// TIA Portal V17 export
// export: Created 2024-09-03T21:55:01.6127892Z, ExportSetting WithDefaults, DisplayName Totally Integrated Automation Portal, DisplayVersion V17 Update 7, DisplayName TIA Portal Openness, DisplayVersion V17 Update 7, DisplayName TIA Portal Version Control Interface, DisplayVersion V17, DisplayName SINAMICS Startdrive Advanced, DisplayVersion V17 SP2, DisplayName SINAMICS Startdrive G110M, G120, G120C, G120D, G120P, G115D, DisplayVersion V17 SP2, DisplayName SINAMICS Startdrive G130, G150, S120, S150, SINAMICS MV, S210, DisplayVersion V17 SP2, DisplayName STEP 7 Professional, DisplayVersion V17 Update 7, DisplayName STEP 7 Safety, DisplayVersion V17 Update 6, DisplayName WinCC Advanced / Unified PC, DisplayVersion V17 Update 7
DATA_BLOCK "IJC_DB"   // DB800
VERSION : 0.1
// stored: AutoNumber false, DBAccessibleFromOPCUA true, DBAccessibleFromWebserver true, InstanceOfName FB_IJC, InstanceOfType FB
"FB_IJC"
   // VAR
   //    MSG { S7_SetPoint := 'True'} : Array[0..30] of "IJC PROTOCOL";
   //    NFP_1 { S7_SetPoint := 'True'} : String[8];
   //    Component_1 : String[30];
   //    NFP_2 : String[8];
   //    Component_2 : String[30];
   //    Send_STA : Array[0..5] of Bool;
   //    Send_TRC : Array[0..5] of Bool;
   //    Send_TRR : Array[0..5] of Bool;
   //    Send_CNF : Array[0..5] of Bool;
   //    IJC_STA_1_Ans_OK : Bool;
   //    IJC_STA_1_Ans_NOK : Bool;
   //    IJC_TRC_1_Ans_OK : Bool;
   //    IJC_TRC_1_Ans_NOK : Bool;
   //    IJC_STA_2_Ans_NOK : Bool;
   //    IJC_STA_2_Ans_OK : Bool;
   //    IJC_TRC_2_Ans_OK : Bool;
   //    IJC_TRC_2_Ans_NOK : Bool;
   //    FP1 : Bool;
   //    FP2 : Bool;
   //    FP3 : Bool;
   //    FP4 : Bool;
   //    FP5 : Bool;
   //    FP6 : Bool;
   //    Reset : Bool;
   //    IJC_Enable : Bool;
   //    DN_STA : Array[0..5] of Bool;
   //    DN_TRC : Array[0..5] of Bool;
   //    DN_TRR : Array[0..5] of Bool;
   //    DN_CNF : Array[0..5] of Bool;
   //    INDEX : Int;
   //    ALL_STA_OK : Bool;
   //    AWAKE_SIGNAL_INSTANCE : "AWAKE_SIGNAL";
   // END_VAR
BEGIN
   MSG[1..4].M_TYPE := 'STA';
   MSG[5..8].M_TYPE := 'TRC';
   MSG[9..10].M_TYPE := 'TRR';
   MSG[11..13].M_TYPE := 'CNF';
   MSG[1].M_NBR := 1;
   MSG[2].M_NBR := 2;
   MSG[3].M_NBR := 3;
   MSG[4].M_NBR := 4;
   MSG[5].M_NBR := 5;
   MSG[6].M_NBR := 6;
   MSG[7].M_NBR := 7;
   MSG[8].M_NBR := 8;
   MSG[9].M_NBR := 9;
   MSG[10].M_NBR := 10;
   MSG[11].M_NBR := 11;
   MSG[12].M_NBR := 12;
   MSG[13].M_NBR := 13;
END_DATA_BLOCK
